ABB RobotStudio station: Gofa_socket_station.rsstn

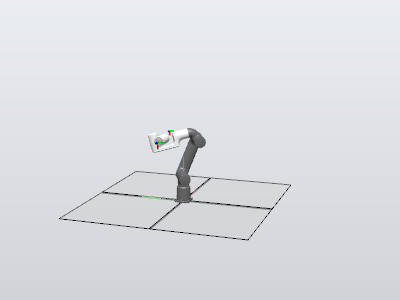
Station Station (saved by RobotStudio 25.2.11220.0)
Controller 15000_real_controller
  mechanical unit ROB_1: CRB15000_5_95__02, 6 joints, base frame (0, 0, 0) mm
Layout (positions relative to the parent item):
  - CRB15000_5_95__02 [mechanism, from %ABB.RobotStudio.Models.CRB15000%\CRB15000_5_95__02.rslib] at (0, 0, 0) mm; joint values [2.0635, -0.3873, 0.6088, -1.4534, -1.0911, 1.3206] (rad or m)
Targets, tools, work objects and paths stored in the station, written as RAPID:
! task T_ROB1
MODULE Corso2806
  PROC mainProva()
    cerchio;
    Rettangolo;
    cerchio;
  ENDPROC
  PROC Rettangolo()
  ENDPROC
  PROC cerchio()
  ENDPROC
ENDMODULE

! task T_ROB1
MODULE TCP_socket
  CONST jointtarget jhome:=[[180,-20,20,0,0,0],[0,9E+09,9E+09,9E+09,9E+09,9E+09]];
  PROC server_recover()
  ENDPROC
  PROC main_socket()
    ConfL \On;
    MoveAbsJ jhome,v500,z50,tool0\WObj:=wobj0;
    WaitTime \InPos,0.1;
    WaitTime \InPos,1;
    WaitTime \InPos,0.1;
    WaitTime \InPos,0.2;
    MoveL rtemp,v1000,z50,tool0\WObj:=wobj0;
    WaitTime \InPos,0.1;
  ENDPROC
ENDMODULE

! task T_ROB1
MODULE ModuleDisassembly
  VAR num ScrewTime:=4;
  PROC Main()
  ENDPROC
  PROC Screw()
    WaitTime ScrewTime;
    WaitTime ScrewTime;
    WaitTime ScrewTime;
    WaitTime ScrewTime;
    WaitTime ScrewTime;
  ENDPROC
ENDMODULE

! task T_ROB1
MODULE Corso0107
  PROC Homing()
    MoveL r_current,v1000,fine,tool0\WObj:=wobj0;
  ENDPROC
  PROC Cerchio_quadrato()
    Homing;
    cechioOffset;
    RettangoloOffset;
  ENDPROC
  PROC Routinereltool()
  ENDPROC
  PROC messaggi2()
    cechioOffset;
    RettangoloOffset;
    Homing;
  ENDPROC
  PROC RettangoloOffset()
  ENDPROC
  PROC messaggi()
    Homing;
    cechioOffset;
    Homing;
  ENDPROC
  PROC cechioOffset()
  ENDPROC
ENDMODULE

